Fanuc KAREL source: CA0071.KL

PROGRAM CA0071
%STACKSIZE=65535
%PRIORITY=65535
%NOLOCKGROUP
VAR
G : INTEGER
I : INTEGER
R : REAL
B : BOOLEAN
S : STRING[16]
AI : ARRAY[2] OF INTEGER
AR : ARRAY[2] OF REAL
P : XYZWPR
-- UNRESOLVED DECLARATIONS (source type spelling not recovered)
-- ST : TYPE_0x1100 (type_u16=0x1100)
-- V : TYPE_0x0013 (type_u16=0x0013)
ROUTINE F(P1 : INTEGER; P2 : REAL; P3 : BOOLEAN; P4 : STRING; P5 : INTEGER; P6 : REAL; P7 : BOOLEAN; P8 : STRING; P9 : INTEGER; P10 : REAL; P11 : BOOLEAN; P12 : STRING; P13 : INTEGER; P14 : REAL; P15 : BOOLEAN; P16 : STRING; P17 : INTEGER;
P18 : REAL; P19 : BOOLEAN; P20 : STRING; P21 : INTEGER; P22 : REAL; P23 : BOOLEAN; P24 : STRING; P25 : INTEGER; P26 : REAL; P27 : BOOLEAN; P28 : STRING; P29 : INTEGER; P30 : REAL; P31 : BOOLEAN; P32 : STRING) FROM CA0071
ROUTINE F
BEGIN
G=(G + 1)
END F
BEGIN
G=0
I=1
R=2.5
B=TRUE
S='A'
AI[1]=3
AR[1]=4.5
ST.A=5
ST.B=1087373312
-- UNSAFE_SOURCE_IR line 64: F(I, ARG_2_UNRESOLVED, B, ARG_4_UNRESOLVED, I, ARG_6_UNRESOLVED, B, ARG_8_UNRESOLVED, I, ARG_10_UNRESOLVED, B, ARG_12_UNRESOLVED, I, ARG_14_UNRESOLVED, B, ARG_16_UNRESOLVED, I, ARG_18_UNRESOLVED, B,
END CA0071
